{attribute 'qualified_only'}
VAR_GLOBAL
	{ attribute 'TcHmiSymbol.AddSymbol' }
	{ attribute 'TcHmiSymbol.ShowRecursively' }
	curingStations:	ARRAY[0..4] OF ST_CURING_STATION_HMI;
	
	{ attribute 'TcHmiSymbol.AddSymbol' }
	{ attribute 'TcHmiSymbol.ShowRecursively' }
	cs:				ST_CS_HMI;
	
	
	csThermo: ST_TIME_PROPORTIONAL_THERMOSTAT_HMI;
END_VAR

(* stored: Version 1.1.0.1
   GVL HMI: Id {d12d1443-11f6-462f-a95b-eab1e526099c} *)
